TEXTLIST LineLoadClase
  0 = '不选择' | Chinese: '不选择' | English: 'None' | Vietnamese: 'None'
  1 = '优先主流线' | Chinese: '优先主流线' | English: 'Priority Line0' | Vietnamese: 'Priority Line0'
  2 = '优先接驳站' | Chinese: '优先接驳站' | English: 'Priority Acquire' | Vietnamese: 'Priority Acquire'
  3 = '优先传感器' | Chinese: '优先传感器' | English: 'Priority Sensor' | Vietnamese: 'Priority Sensor'
   = ''
END_TEXTLIST

(* stored: Version 1.1.0.1, ProductVersion 3.1.4024.3
   TextList LineLoadClase: Id {c338f25a-dd3d-4a81-a9bd-0921cc96e445} *)
